FUNCTION_BLOCK ILOCK_BLOCK_PROTECT_AX (* Prioritizes the first active input with protection dead-time (Adapter Version). *)
  (* Standard: 61499-2; Description: Copyright (c) 2023 HR Agrartechnik GmbH This program and the accompanying materials are made available under the terms of the Eclipse Public License 2.0 which is available at https://www.eclipse.org/legal/epl-2.0/ SPDX-License-Identifier: EPL-2.0 *)
  (* Version 1.2, 2026-04-19, Franz Höpfinger, HR Agrartechnik GmbH, Fixed: Re-added UPDATE event for DT_PROTECT and used it in ECC to satisfy Basic FB rules *)
  PACKAGE logiBUS::signalprocessing::interlock;
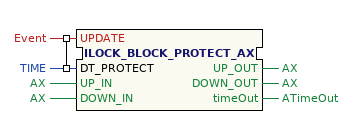
  EVENT_INPUT
    UPDATE WITH DT_PROTECT; (* Update parameters *)
  END_EVENT
  VAR_INPUT
    DT_PROTECT : TIME := T#50ms; (* Protection Time *)
  END_VAR
  SOCKETS
    UP_IN : adapter::types::unidirectional::AX; (* Input for forward/up direction *)
    DOWN_IN : adapter::types::unidirectional::AX; (* Input for backward/down direction *)
  END_SOCKETS
  PLUGS
    UP_OUT : adapter::types::unidirectional::AX; (* Output for forward/up direction *)
    DOWN_OUT : adapter::types::unidirectional::AX; (* Output for backward/down direction *)
    timeOut : iec61499::events::ATimeOut; (* timeOut Adapter *)
  END_PLUGS
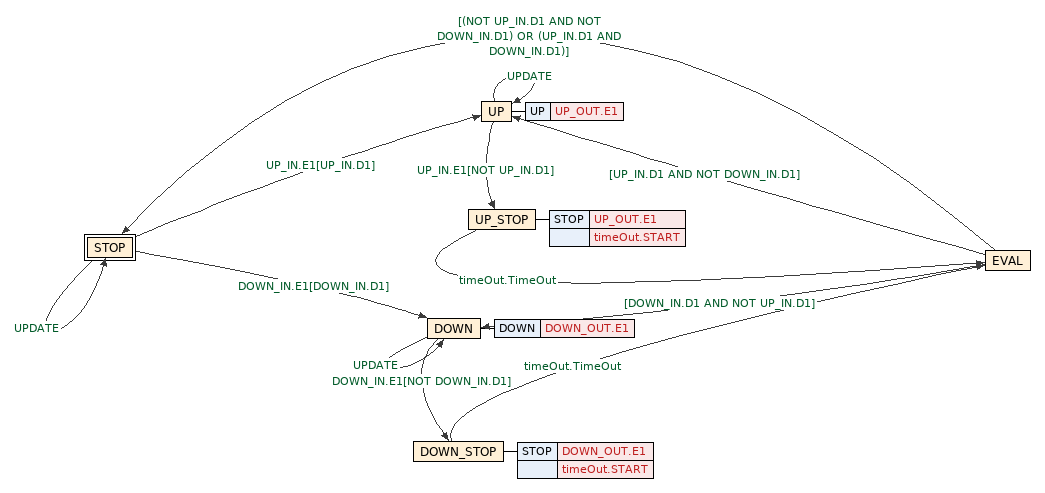
  EC_STATES
    STOP;
    UP : UP -> UP_OUT.E1;
    DOWN : DOWN -> DOWN_OUT.E1;
    UP_STOP : STOP -> UP_OUT.E1, -> timeOut.START;
    DOWN_STOP : STOP -> DOWN_OUT.E1, -> timeOut.START;
    EVAL;
  END_STATES
  EC_TRANSITIONS
    STOP TO DOWN := DOWN_IN.E1[DOWN_IN.D1];
    STOP TO UP := UP_IN.E1[UP_IN.D1];
    DOWN TO DOWN_STOP := DOWN_IN.E1[NOT DOWN_IN.D1];
    UP TO UP_STOP := UP_IN.E1[NOT UP_IN.D1];
    UP_STOP TO EVAL := timeOut.TimeOut;
    DOWN_STOP TO EVAL := timeOut.TimeOut;
    EVAL TO UP := [UP_IN.D1 AND NOT DOWN_IN.D1];
    EVAL TO DOWN := [DOWN_IN.D1 AND NOT UP_IN.D1];
    EVAL TO STOP := [(NOT UP_IN.D1 AND NOT DOWN_IN.D1) OR (UP_IN.D1 AND DOWN_IN.D1)];
    STOP TO STOP := UPDATE;
    UP TO UP := UPDATE;
    DOWN TO DOWN := UPDATE;
  END_TRANSITIONS
  ALGORITHM UP IN ST:
timeOut.DT := DT_PROTECT;
UP_OUT.D1 := BOOL#TRUE;
DOWN_OUT.D1 := BOOL#FALSE;
  END_ALGORITHM
  ALGORITHM DOWN IN ST:
timeOut.DT := DT_PROTECT;
UP_OUT.D1 := BOOL#FALSE;
DOWN_OUT.D1 := BOOL#TRUE;
  END_ALGORITHM
  ALGORITHM STOP IN ST:
timeOut.DT := DT_PROTECT;
UP_OUT.D1 := BOOL#FALSE;
DOWN_OUT.D1 := BOOL#FALSE;
  END_ALGORITHM
END_FUNCTION_BLOCK
